FUNCTION_BLOCK FB_06_ExSTOP
VAR_INPUT
	bExecute:BOOL;
END_VAR
VAR_OUTPUT
	bBusy:BOOL;(*功能块执行忙标志*)
	bError:BOOL;(*出错*)
	bDone:BOOL;(*执行完毕*)
END_VAR
VAR_IN_OUT
//	stX:AXIS_REF;
//	stY:AXIS_REF;
//	stZ:AXIS_REF;
	stItpToPlc :NCTOPLC_NCICHANNEL_REF;
	stPlcToItp:PLCTONC_NCICHANNEL_REF;
END_VAR
VAR
	StopStep:INT:=0;
	fbEStop:ItpEStopEx;(*暂停*)
END_VAR

CASE StopStep OF
	0:
	  IF  bExecute THEN
		 bBusy:=TRUE;(*FB执行状态*)
		 bDone:=FALSE;(*FB执行完毕*)
		 bError:=FALSE;(*报错*)
		 StopStep:=10;(*进入10步*) 
	  END_IF
	10:
	  fbEStop(
	    sNciToPlc:=stItpToPlc , 
	    bExecute:= TRUE, 
	    fDec:= 40000, 
	    fJerk:= 40000, 
	    tTimeOut:= , 
	    bBusy=> , 
	    bErr=> , 
	    nErrId=> );
	   IF NOT fbEStop.bBusy THEN
		  IF NOT fbEStop.bErr THEN
			StopStep:=20;(*进入20步*)  
		  ELSE
			bBusy:=FALSE;
			bError:=TRUE;
			StopStep:=999;
		  END_IF
		  fbEStop(bExecute:= FALSE,sNciToPlc:= stItpToPlc); 
	    END_IF
	 20:
	   bDone:=TRUE;
       bBusy:=FALSE;   
	   IF NOT bExecute THEN
		 StopStep:=0;
	   END_IF
	 999:
	   IF NOT bExecute THEN		   
	    StopStep:=0;
        bError:=FALSE; 
	   END_IF
END_CASE

END_FUNCTION_BLOCK

(* stored: Version 1.1.0.1, ProductVersion 3.1.4024.12
   POU FB_06_ExSTOP: Id {ad22736d-bf35-424d-8035-d5e51fcbc6c9}, SpecialFunc None *)
